FUNCTION_BLOCK SludgeBufferSensors (* Composite Function Block Type *)
  (* Standard: 61499-2 *)
  (* Version 0.0, 7/1/2024, NVPP, Schneider Electric, template *)
  PACKAGE SE.Nereda;
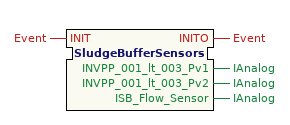
  EVENT_INPUT
    INIT;
  END_EVENT
  EVENT_OUTPUT
    INITO;
  END_EVENT
  PLUGS
    INVPP_001_lt_003_Pv1 : IAnalog; (* Process value and status interface adapter *)
    INVPP_001_lt_003_Pv2 : IAnalog; (* Process value and status interface adapter *)
    ISB_Flow_Sensor : IAnalog; (* Process value and status interface adapter *)
  END_PLUGS
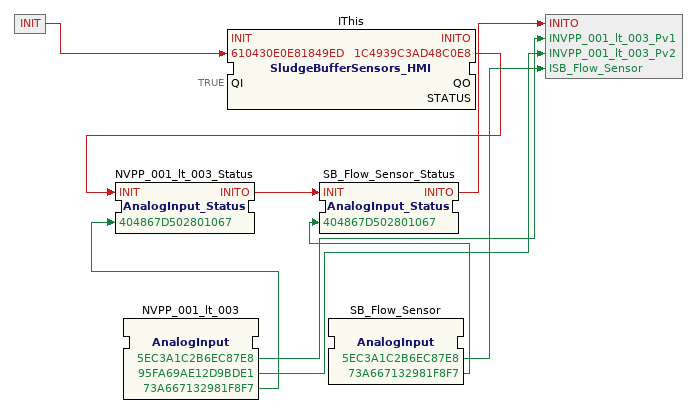
  (* 01 - FUNCTIONNAL INPUT INTERFACE *)
  (* 00 - INITIALIZATION *)
  (* 06 - HMI INTERFACE *)
  (* 02 - FUNCTIONNAL OUTPUT INTERFACE *)
  (* 03 - FIELD INTERFACE *)
  (* Level measurement sludge buffer *)
  (* Pressure sensor 2 *)
  (* 05 - LOGIC *)
  (* Actuators Status *)
  FBS
    IThis : SludgeBufferSensors_HMI(QI := TRUE);
    NVPP_001_lt_003 : AnalogInput;
    SB_Flow_Sensor : AnalogInput;
    NVPP_001_lt_003_Status : AnalogInput_Status;
    SB_Flow_Sensor_Status : AnalogInput_Status;
  END_FBS
  EVENT_CONNECTIONS
    INIT TO IThis.610430E0E81849ED;
    NVPP_001_lt_003_Status.INITO TO SB_Flow_Sensor_Status.INIT;
    IThis.1C4939C3AD48C0E8 TO NVPP_001_lt_003_Status.INIT;
    SB_Flow_Sensor_Status.INITO TO INITO;
  END_CONNECTIONS
  ADAPTER_CONNECTIONS
    NVPP_001_lt_003.5EC3A1C2B6EC87E8 TO INVPP_001_lt_003_Pv1;
    NVPP_001_lt_003.95FA69AE12D9BDE1 TO INVPP_001_lt_003_Pv2;
    SB_Flow_Sensor.5EC3A1C2B6EC87E8 TO ISB_Flow_Sensor;
    NVPP_001_lt_003.73A667132981F8F7 TO NVPP_001_lt_003_Status.404867D502801067;
    SB_Flow_Sensor.73A667132981F8F7 TO SB_Flow_Sensor_Status.404867D502801067;
  END_CONNECTIONS
END_FUNCTION_BLOCK
